PROGRAM MAIN
VAR
pwmInstance : FB_PWM;
END_VAR

pwmInstance(fPeriod := 1000, fDutyCycle := 50); // Voorbeeldwaarden

END_PROGRAM

(* stored: Version 1.1.0.1, ProductVersion 3.1.4024.12
   POU MAIN: Id {f7236189-f2e9-4dfb-a883-e9d30d96e06e}, SpecialFunc None *)
